{attribute addProperty BoxType "EJ7041-0052-0016"}
{attribute addProperty Id "ENC_Status_compactAT %I*ENC_Status_compact_FA080ECA4860STM_StatusAT %I*STM_Status_64D937431620ENC_Control_compactAT %Q*ENC_Control_compact_5C86AA9D3240STM_ControlAT %Q*STM_Control_6F24B2C41620STM_VelocityAT %Q*STM_Velocity_1D89B5C21620WcStateAT %I*WcState_F855686C1620InfoDataAT %I*InfoData_1C46E3E796120"}
{attribute addProperty CRC "2903822255"}
{attribute addProperty SizeInBites "240"}
{attribute addProperty SizeInBytes "30"}
TYPE EJ7041_61C571CF :
STRUCT
	{attribute addProperty Name "ENC_Status_compact"}
	ENC_Status_compact : ENC_Status_compact_FA080ECA;
	{attribute addProperty Name "STM_Status"}
	STM_Status : STM_Status_64D93743;
	{attribute addProperty Name "ENC_Control_compact"}
	ENC_Control_compact : ENC_Control_compact_5C86AA9D;
	{attribute addProperty Name "STM_Control"}
	STM_Control : STM_Control_6F24B2C4;
	{attribute addProperty Name "STM_Velocity"}
	STM_Velocity : STM_Velocity_1D89B5C2;
	{attribute addProperty Name "WcState"}
	WcState : WcState_F855686C;
	{attribute addProperty Name "InfoData"}
	InfoData : InfoData_1C46E3E7;
END_STRUCT
END_TYPE

(* stored: Version 1.2.0.0, ProductVersion 3.1.4024.9
   DUT EJ7041_61C571CF: Id {c95f29af-cef3-4fd6-a768-60163a4d1bc4} *)
